PROGRAM POU_VisButton
VAR
	
xUp	:	BOOL;
xDown	:	BOOL;

yUp	:	BOOL;
yDown	:	BOOL;

zuP	:	BOOL;	
zDown	:	BOOL;

DecVal	:	LREAL;



	xUpR_TRIG: R_TRIG;
	xDownR_TRIG: R_TRIG;
	yUpR_TRIG: R_TRIG;
	yDownR_TRIG: R_TRIG;
	zUpR_TRIG: R_TRIG;
	zDownR_TRIG: R_TRIG;
	BridgeValZ: LREAL;
END_VAR

	
xUpR_TRIG(CLK:=xUp , Q=> );
xDownR_TRIG(CLK:=xDown , Q=> );

yUpR_TRIG(CLK:=yUp , Q=> );
yDownR_TRIG(CLK:=yDown , Q=> );

zUpR_TRIG(CLK:=zUp , Q=> );
zDownR_TRIG(CLK:=zDown , Q=> );


stAxisZ.In.fSetPos	:=	BridgeValZ;

	//stAxisX.In.fSetPos;
	//stAxisY.In.fSetPos;
	//stAxisZ.In.fSetPos;

IF xUpR_TRIG.Q	THEN
	
stAxisX.In.fSetPos	:=	stAxisX.In.fSetPos	+	10;


ELSIF xDownR_TRIG.Q THEN
	stAxisX.In.fSetPos	:=	stAxisX.In.fSetPos	-	10;
END_IF



IF yUpR_TRIG.Q	THEN
	
stAxisY.In.fSetPos	:=	stAxisY.In.fSetPos	+	10;


ELSIF yDownR_TRIG.Q THEN
	stAxisY.In.fSetPos	:=	stAxisY.In.fSetPos	-	10;
END_IF




IF zUpR_TRIG.Q	THEN
	
BridgeValZ	:=	BridgeValZ	+	10;


ELSIF zDownR_TRIG.Q THEN
	BridgeValZ	:=	BridgeValZ	-	10;
END_IF

END_PROGRAM

(* stored: Version 1.1.0.1, ProductVersion 3.1.4024.0
   POU POU_VisButton: Id {7681f85b-4e97-401a-83c7-d4bd560bd69e}, SpecialFunc None *)
